INTERFACE I_HE_SATT_Filter EXTENDS __System.IQueryInterface


PROPERTY Holder : I_HE_SATT_FilterHolder
GET
END_GET
END_PROPERTY


PROPERTY Length : LREAL
GET
END_GET
END_PROPERTY


PROPERTY Material : E_HE_SATT_FilterMaterial
GET
END_GET
END_PROPERTY

PROPERTY MaterialFormula : T_MaxString
GET
END_GET
END_PROPERTY

PROPERTY Status : E_HE_SATT_FilterStatus
GET
END_GET
END_PROPERTY

END_INTERFACE

(* stored: Version 1.1.0.1
   Itf I_HE_SATT_Filter: Id {bd19a689-7463-44af-b072-8b6f73cd8774}
   Property Holder: Id {d8427123-d076-4c33-81b3-e42e5841a1a7}
   Get Get: Id {6bd88ea0-16ab-446f-83ea-d28b5c458d10}
   Property Length: Id {950ec1a2-9429-4ffc-bb31-b4743299bd35}
   Get Get: Id {214889b9-0f87-4344-af90-850efc1dac34}
   Property Material: Id {643cb2d7-b5cb-4b11-900a-64fe1430e86c}
   Get Get: Id {88a78f22-035c-4585-aec5-e6783836e3bd}
   Property MaterialFormula: Id {9e7d0162-9d6f-4bea-9492-8ee2a77816ee}
   Get Get: Id {d290165d-4fbf-45a0-af70-49c51bd8a6e3}
   Property Status: Id {bb6a4b26-2f02-4902-83bb-232dfe0204b2}
   Get Get: Id {6f954fc4-8797-4be2-b028-5988ed9b6329} *)
